FUNCTION_BLOCK FB_Position
VAR
	_X : LREAL;
	_Y : LREAL;
END_VAR

PROPERTY PosXY : S_PosXY
GET
PosXY.X := _X;
PosXY.Y := _Y;
END_GET
SET
_X := PosXY.X;
_Y := PosXY.Y;
END_SET
END_PROPERTY

METHOD SetXY : S_PosXY
VAR_INPUT
	X : LREAL;
	Y : LREAL;
END_VAR
_X := X;
_Y := Y;
SetXY.X := _X;
SetXY.Y := _Y;
END_METHOD

PROPERTY X : LREAL
GET
X:=_X;
END_GET
SET
_X:=X;
END_SET
END_PROPERTY

PROPERTY Y : LREAL
GET
Y:=_Y;
END_GET
SET
_Y:=Y;
END_SET
END_PROPERTY

END_FUNCTION_BLOCK

(* stored: Version 1.1.0.1
   POU FB_Position: Id {f7738b07-0372-4fa3-ab31-108d17739e14}, SpecialFunc None
   Property PosXY: Id {bcc072ae-c9cb-4529-adb0-d581ffb64fe6}
   Get Get: Id {5cf5a3f0-9869-41ba-bd38-b8024da122ac}
   Set Set: Id {af967654-a4fd-4523-9184-79289696139b}
   Method SetXY: Id {63ce22ec-eb8a-4ce5-87a6-3e3eb833289b}
   Property X: Id {1a8ba78a-663d-4c79-a09c-adcc8858c283}
   Get Get: Id {7443a80b-3097-4227-8eef-f1665863793f}
   Set Set: Id {c8019f09-c635-46c0-b7fd-e448cbe7d3b9}
   Property Y: Id {c30cff65-c3a6-4814-b85f-3d90b2df0457}
   Get Get: Id {f900bc93-ad24-4f26-9a61-dc679bfe1240}
   Set Set: Id {2d3b4512-edc0-4c3c-88a1-a7e9fe6c77e7} *)
